{attribute addProperty BoxType "EK1100-0000-0018"}
{attribute addProperty Id "Beckhoff_EQ3xxxEK1122Beckhoff_EQ3xxxEK1122_C2B88B713460432.5"}
{attribute addProperty CRC "466567580"}
{attribute addProperty SizeInBites "3460"}
{attribute addProperty SizeInBytes "432.5"}
TYPE Beckhoff_EQ3xxx_1BCF419C EXTENDS EK1100_179A0949 :
STRUCT
	{attribute addProperty Name "Beckhoff_EQ3xxxEK1122"}
	Beckhoff_EQ3xxxEK1122 : Beckhoff_EQ3xxxEK1122_C2B88B71;
END_STRUCT
END_TYPE

(* stored: Version 1.2.0.0, ProductVersion 3.1.4024.9
   DUT Beckhoff_EQ3xxx_1BCF419C: Id {80c4fce9-ad2c-4ed5-90e9-dfaf35a59271} *)
